PROGRAM MAIN
VAR
END_VAR

END_PROGRAM

(* stored: Version 1.1.0.1
   POU MAIN: Id {86273dcd-f42f-437d-8c99-a1e944cf788a} *)
